{attribute addProperty BoxType "BK1120-0000-0019"}
{attribute addProperty Id "Term_379_KL1002KL1002_D229A9CA00"}
{attribute addProperty CRC "554172164"}
{attribute addProperty SizeInBites "0"}
{attribute addProperty SizeInBytes "0"}
TYPE A_0006_BK1120_0000_0019_2107FF04 EXTENDS BK1120_4487A81F :
STRUCT
	{attribute addProperty Name "Term_379_KL1002"}
	Term_379_KL1002 : KL1002_D229A9CA;
END_STRUCT
END_TYPE

(* stored: Version 1.2.0.0, ProductVersion 3.1.4024.9
   DUT A_0006_BK1120_0000_0019_2107FF04: Id {18598ee0-6339-4048-b3c1-95405ed0962e} *)
